PROGRAM MAIN
VAR
END_VAR

PRG_DIAGNOSTIC();
PRG_GMD();

END_PROGRAM

(* stored: Version 1.1.0.1, ProductVersion 3.1.4022.12
   POU MAIN: Id {1b83c7bd-a799-4af4-95bc-f736ed100852}, SpecialFunc None *)
